FUNCTION F_UpdateParametersByReference : LREAL
VAR_INPUT
	bSetNewValue : BOOL;
	fMaxPistonStroke : LREAL;
	paramCylinderPiston : REFERENCE TO ST_pPistonRange;
END_VAR
VAR

END_VAR

IF bSetNewValue THEN
	paramCylinderPiston.fPistonPosMax := fMaxPistonStroke;
	bSetNewValue := FALSE;
END_IF

END_FUNCTION

(* stored: Version 1.1.0.1, ProductVersion 3.1.4024.10
   POU F_UpdateParametersByReference: Id {4beb6302-9d61-4873-b93a-92b401a4fe4c}, SpecialFunc None *)
